// Block: PPrgArchive4

DATA_BLOCK PPrgArchive4
VERSION : 0.1
   NON_RETAIN
   VAR
      PRG : Array[301..400] of PPrg_Data;
   END_VAR

BEGIN
   // No initialization required
END_DATA_BLOCK
